// TIA Portal V17 export
// export: Created 2024-09-27T18:48:47.1351468Z, ExportSetting WithDefaults, DisplayName Totally Integrated Automation Portal, DisplayVersion V17, DisplayName TIA Portal Openness, DisplayVersion V17, DisplayName TIA Portal Version Control Interface, DisplayVersion V17, DisplayName STEP 7 Professional, DisplayVersion V17, DisplayName STEP 7 Safety, DisplayVersion V17, DisplayName WinCC Professional, DisplayVersion V17
DATA_BLOCK "MC_Power_DB"   // DB9
// stored: AutoNumber true, DBAccessibleFromOPCUA true, InstanceOfName MC_Power, OfSystemLibElement MC_Power, OfSystemLibVersion 8.0
"MC_Power"
   // VAR_INPUT
   //    Axis : TO_Axis;
   //    Enable : Bool;
   //    StartMode : Int;
   //    StopMode : Int;
   // END_VAR
   // VAR_OUTPUT
   //    Status : Bool;
   //    Busy : Bool;
   //    Error : Bool;
   //    ErrorID : Word;
   //    ErrorInfo : Word;
   // END_VAR
   // VAR
   //    FB_ID : DInt;
   // END_VAR
BEGIN
END_DATA_BLOCK
